# EPICS autosave request: 3-0/iocBoot/iocAMC100Test/AMC100Test_settings.req
# scan and SaveData settings
file standardScans_settings.req P=$(IOC)
file saveData_settings.req P=$(IOC)

# Controller settings that motorRecord does not support
file "amc100_dmc_ctrl.req" P=$(P)

# Motor record settings
# Real motors
file "motor_settings.req" P=$(P), M=MTR1
file "motor_settings.req" P=$(P), M=MTR2
file "motor_settings.req" P=$(P), M=MTR3

file "amc100_motor_settings.req" P=$(P), M=MTR1
file "amc100_motor_settings.req" P=$(P), M=MTR2
file "amc100_motor_settings.req" P=$(P), M=MTR3
